TYPE ST_XPU_STRINGS :
STRUCT
  sXpuState       ,
  sXpuResult      ,
  sXpuCyclicCheck ,
  sXpuOpMode      ,
  sXpuMoverId_DetectionMode,
  sXpuMoverPosAssignement : STRING(30) := 'NULL';
END_STRUCT
END_TYPE

(* stored: Version 1.1.0.1, ProductVersion 3.1.4026.13
   DUT ST_XPU_STRINGS: Id {214fa312-1e18-4fe5-8e85-595059d28eed} *)
